(* IEC 61131-3 sources: programs/VI-54/VI-54_20171205/VI-54_20171205/Stations/Screen/LseClass170718/Class/USBDetection, 1 file *)

(* ---- USBDetection.st ---- *)
#define USB_StringLength                              _strlen("C:\")          // Länge des Strings für das aktuelle Laufwerk

(*!
<Class
	Name               = "USBDetection"
	Revision           = "1.2"
	RealtimeTask       = "false"
	CyclicTask         = "false"
	BackgroundTask     = "false"
	Sigmatek           = "false"
	OSInterface        = "false"
	HighPriority       = "false"
	Automatic          = "false"
	UpdateMode         = "Prescan"
	SharedCommandTable = "true"
	Objectsize         = "(540,360)"
	Comment            = "class detects a plugged USB device (USBdetected) &#13;&#10;and writes it&apos;s drive letter to a string object">
	<Channels>
		<Server Name="DriveIndex" Visualized="false" Initialize="false" WriteProtected="false" Retentive="false" Comment="internal index of the plugged USB device"/>
		<Server Name="DriveLetter" Class="String" Visualized="false" Initialize="true" WriteProtected="false" Retentive="false" Comment="drive letter of the plugged USB device  &#13;&#10;&quot;C:\&quot;: means that NO USB device is detected "/>
		<Server Name="DriveListError" Visualized="false" Initialize="false" WriteProtected="true" Retentive="false" Comment="1= function GetDriveListShort failed"/>
		<Server Name="USBdetected" Visualized="true" Initialize="false" WriteProtected="false" Retentive="false" Comment="0= no USB device found&#13;&#10;1= USB device is plugged"/>
		<Client Name="FileSys" Required="false" Internal="false" Comment="object channel to FileSys (don&apos;t connect)"/>
		<Client Name="USBDriveLetter" Required="true" Internal="true"/>
	</Channels>
	<RevDoku>
		<Owner Company="Sigmatek" Author="BraLis"/>
		<Dokumentation Revision="1.2&#13;&#10;" Date="2015-09-23" Author="BraLis" Company="Sigmatek" Description="the client coDriveLetter from the class AccessControlMain was connected wrongly, now connected with the server DriveLetter from the class USBDetection"/>
		<Dokumentation Revision="1.1" Date="2015-09-22" Company="Sigmatek" Description="Creation."/>
	</RevDoku>
	<Network Name="USBDetection">
		<!-- List of Components in this network -->
		<Components>
			<Object
				Name       = "_base"
				Class      = "_Global"
				Position   = "(218,120)"
				Visualized = "false">
				<Channels>
					<Server Name="Server0"/>
					<Client Name="Lse"/>
				</Channels>
			</Object>
			<Object
				Name       = "USBDriveLetter"
				Class      = "String"
				Position   = "(240,300)"
				Visualized = "true">
				<Channels>
					<Server Name="Data"/>
					<Client Name="SingleRealloc" Value="1"/>
				</Channels>
			</Object>
		</Components>
		<Comments>
		</Comments>
		<!-- List of Connections in this network -->
		<Connections>
			<Connection Source="this.Server0" Destination="_base.Server0" Vertices="(968,210),(518,210),"/>
			<Connection Source="_base.Lse" Destination="this.Lse" Vertices="(218,210),(38,210),"/>
			<Connection Source="this.USBDriveLetter" Destination="USBDriveLetter.Data"/>
			<Connection Source="this.DriveLetter" Destination="USBDriveLetter.Data" Vertices="(968,390),(796,390),"/>
		</Connections>
		<!-- Headerfiles -->
		<Options>
		</Options>
	</Network>
</Class>
*)
#pragma using _Global

USBDetection : CLASS
: _Global
	TYPE
	  Letters :
	  (
	    _A,
	    _B,
	    _C,
	    _D,
	    _E,
	    _F,
	    _G,
	    _H,
	    _I,
	    _J,
	    _K,
	    _L,
	    _M,
	    _N,
	    _O,
	    _P,
	    _Q,
	    _R,
	    _S,
	    _T,
	    _U,
	    _V,
	    _W,
	    _X,
	    _Y,
	    _Z
	  )$UDINT;
	END_TYPE
  //Servers:
	USBdetected 	: SvrCh_DINT;
	DriveListError 	: SvrCh_DINT;
	DriveLetter 	: SvrChCmd_UDINT;
	DriveIndex 	: SvrCh_DINT;
  //Clients:
	FileSys 	: CltChCmd__FileSys;
	USBDriveLetter 	: CltChCmd_String;
  //Variables:
		DriveList : ARRAY [0..25] OF CHAR;

		udUSBdetected 	: UDINT;
  //Functions:

	FUNCTION VIRTUAL GLOBAL Init;

	FUNCTION VIRTUAL GLOBAL IF_WindowRun
		VAR_INPUT
			whoami 	: ^_WHOAMI;
			pic 	: ^void;
			event 	: ^_EVENT;
		END_VAR;
				//! <Function Comment="Sets the server DriveLetter, based on the data from the Drivelist." Name="GetDriveLetter"/>
	FUNCTION GLOBAL GetDriveLetter;
				//! <Function Comment="Gets the data for the Drivelist." Name="GetDriveListInfo"/>
	FUNCTION VIRTUAL GLOBAL GetDriveListInfo;

	FUNCTION VIRTUAL GLOBAL DriveLetter::Read
		VAR_OUTPUT
			output (EAX) 	: UDINT;
		END_VAR;

	FUNCTION VIRTUAL GLOBAL DriveLetter::Write
		VAR_INPUT
			input (EAX) 	: UDINT;
		END_VAR
		VAR_OUTPUT
			result (EAX) 	: UDINT;
		END_VAR;
  //Tables:
	FUNCTION @STD
		VAR_OUTPUT
			ret_code	: CONFSTATES;
		END_VAR;
	FUNCTION GLOBAL TAB @CT_;
END_CLASS;

#pragma using String
#pragma usingLtd _FileSys

FUNCTION VIRTUAL GLOBAL USBDetection::Init

  if _FirstScan then

    // Methode der Basis-Klasse aufrufen
    _Global::init();

    USBDriveLetter.WriteDataOff(USB_StringLength, 0, "C:\");

  end_if;

END_FUNCTION

FUNCTION VIRTUAL GLOBAL USBDetection::IF_WindowRun
	VAR_INPUT
		whoami  : ^_WHOAMI;
		pic 	  : ^void;
		event 	: ^_EVENT;
	END_VAR

  // Methode der Basis-Klasse aufrufen
  _Global::IF_WindowRun(whoami, pic, event);

  // Ereignis am USB-Port aufgetreten?
  if event^.ftype <> _EVENT_NONE then
    if (event^.ftype = _EVENT_LASALOS) & (event^.scancode = 8)then

      // USB-Stick eingesteckt
      //-----------------------------------------------------------------------------------------
      if event^.modifier = 1 then

        // Index des Laufwerksbuchstaben des USB-Sticks
        GetDriveListInfo();

        // setze den Server USBdetected auf 1, wenn ein USB-Stick erkannt wurde
        USBdetected := 1;

        //*****************************************************************************
        //** setze den Pfad laut dem Index des Laufwerksbuchstaben des USB-Sticks    **
        //*****************************************************************************
        case udUSBdetected of

          0:  USBDriveLetter.WriteDataOff(USB_StringLength, 0, "A:\");

          1:  USBDriveLetter.WriteDataOff(USB_StringLength, 0, "B:\");

          3:  USBDriveLetter.WriteDataOff(USB_StringLength, 0, "D:\");

          4:  USBDriveLetter.WriteDataOff(USB_StringLength, 0, "E:\");

          5:  USBDriveLetter.WriteDataOff(USB_StringLength, 0, "F:\");

          6:  USBDriveLetter.WriteDataOff(USB_StringLength, 0, "G:\");

          7:  USBDriveLetter.WriteDataOff(USB_StringLength, 0, "H:\");

          8:  USBDriveLetter.WriteDataOff(USB_StringLength, 0, "I:\");

          9:  USBDriveLetter.WriteDataOff(USB_StringLength, 0, "J:\");

          10: USBDriveLetter.WriteDataOff(USB_StringLength, 0, "K:\");

          11: USBDriveLetter.WriteDataOff(USB_StringLength, 0, "L:\");

          12: USBDriveLetter.WriteDataOff(USB_StringLength, 0, "M:\");

          13: USBDriveLetter.WriteDataOff(USB_StringLength, 0, "N:\");

          14: USBDriveLetter.WriteDataOff(USB_StringLength, 0, "O:\");

          15: USBDriveLetter.WriteDataOff(USB_StringLength, 0, "P:\");

          16: USBDriveLetter.WriteDataOff(USB_StringLength, 0, "Q:\");

          17: USBDriveLetter.WriteDataOff(USB_StringLength, 0, "R:\");

          18: USBDriveLetter.WriteDataOff(USB_StringLength, 0, "S:\");

          19: USBDriveLetter.WriteDataOff(USB_StringLength, 0, "T:\");

          20: USBDriveLetter.WriteDataOff(USB_StringLength, 0, "U:\");

          21: USBDriveLetter.WriteDataOff(USB_StringLength, 0, "V:\");

          22: USBDriveLetter.WriteDataOff(USB_StringLength, 0, "W:\");

          23: USBDriveLetter.WriteDataOff(USB_StringLength, 0, "X:\");

          24: USBDriveLetter.WriteDataOff(USB_StringLength, 0, "Y:\");

          25: USBDriveLetter.WriteDataOff(USB_StringLength, 0, "Z:\");

        end_case;

      // USB-Stick entfernt
      //-----------------------------------------------------------------------------------------
      elsif event^.modifier = 2 then

        // setze den Server USBdetected auf 0, wenn kein USB-Stick erkannt wurde
        USBdetected := 0;

        USBDriveLetter.WriteDataOff(USB_StringLength, 0, "C:\");

      end_if;

    end_if;
  end_if;

END_FUNCTION

FUNCTION VIRTUAL GLOBAL USBDetection::GetDriveListInfo
  VAR
    State   : DINT;
  END_VAR

  // hole Daten der DriveList
  State := FileSys.GetDriveListShort(drivelist:= #DriveList$CHAR);

  // setze DriveListError wenn kein Speichermedium existiert
  if State <> 0 then
    DriveListError := 1;
  end_if;

  // hole den Index eines Speichermediums
  GetDriveLetter();

END_FUNCTION

FUNCTION GLOBAL USBDetection::GetDriveLetter
  VAR
    i   : UDINT;
  END_VAR

  for i:=0 to 25 do
    // überspringe "C:\\"
    if i <> 2 then

      // suche nach dem Index eines Speichermediums
      if (Drivelist[i] <> 16#00) then

        // speichere den letzten Index
        udUSBdetected := i;

        DriveIndex.Write(input:=to_dint(i));

      end_if;

    end_if;
  end_for;

END_FUNCTION

FUNCTION VIRTUAL GLOBAL USBDetection::DriveLetter::Read
	VAR_OUTPUT
		output (EAX) 	: UDINT;
	END_VAR

	DriveLetter := USBDriveLetter.Data.Read();
	output := DriveLetter;

END_FUNCTION

FUNCTION VIRTUAL GLOBAL USBDetection::DriveLetter::Write
	VAR_INPUT
		input (EAX) 	: UDINT;
	END_VAR
	VAR_OUTPUT
		result (EAX) 	: UDINT;
	END_VAR

	DriveLetter := input;
	result := (USBDriveLetter.Data.Write(DriveLetter))$UDINT;

END_FUNCTION
